// TwinCAT 3 PLC project WeldApp
// ProgramVersion: 3.1.4024.0
// libraries:
//   Tc2_Standard, * (Beckhoff Automation GmbH)
//   Tc2_System, * (Beckhoff Automation GmbH)
//   Tc3_Module, * (Beckhoff Automation GmbH)
//   VisuDialogs, * (System)
// project tree:
//   DUTs/ FixtureInput.TcDUT (not stored), FixtureOutput.TcDUT, Fixture_Clamp.TcDUT
//   / GlobalTextList.TcGTLO, PlcTask.TcTTO, Visualization Manager.TcVMO (not stored)
//   GVLs/ IO.TcGVL, IO_1.TcGVL, IO_1_1.TcGVL, IO_2.TcGVL
//   POUs/ FB_AutoSequence.TcPOU, FB_Clamp.TcPOU, FB_Robot_MH.TcPOU, FB_RollerDoor.TcPOU, FB_ModeManager.TcPOU, FB_Robot.TcPOU, MAIN.TcPOU, FB_Trunnion.TcPOU, FB_TurnTable.TcPOU, TextList_State1.TcTLO, TextList_State2.TcTLO, Visualization.TcVIS
// real-time tasks:
//   TASK PlcTask: cycle T#10ms, priority 20, ADS port 350

CONFIGURATION WeldApp
    RESOURCE PLC ON TwinCAT3
        TASK PlcTask(INTERVAL := T#10ms, PRIORITY := 20);
        PROGRAM MAIN WITH PlcTask : MAIN;
    END_RESOURCE
END_CONFIGURATION

// ---- DUTs/FixtureOutput.TcDUT
TYPE FixtureOutput :
STRUCT
o_CC1_CLAMPING_UNIT1_3_WP:BOOL;
o_CC1_CLAMPING_UNIT1_3_HP:BOOL;
o_CC2_CLAMPING_UNIT2_3_WP:BOOL;
o_CC2_CLAMPING_UNIT2_3_HP:BOOL;
o_CC3_CLAMPING_UNIT3_3_WP:BOOL;
o_CC3_CLAMPING_UNIT3_3_HP:BOOL;
o_CC4_CLAMPING_UNIT4_3_WP:BOOL;
o_CC4_CLAMPING_UNIT4_3_HP:BOOL;
o_CC5_CLAMPING_UNIT5_1_WP:BOOL;
o_CC5_CLAMPING_UNIT5_1_HP:BOOL;
o_CC6_CLAMPING_UNIT6_1_WP:BOOL;
o_CC6_CLAMPING_UNIT6_1_HP:BOOL;
o_RESERVE_1_4:BOOL;
o_RESERVE_1_5:BOOL;
o_RESERVE_1_6:BOOL;
o_RESERVE_1_7:BOOL;
o_RESERVE_2_0:BOOL;
o_RESERVE_2_1:BOOL;
o_RESERVE_2_2:BOOL;
o_RESERVE_2_3:BOOL;
o_RESERVE_2_4:BOOL;
o_RESERVE_2_5:BOOL;
o_RESERVE_2_6:BOOL;
o_RESERVE_2_7:BOOL;
o_RESERVE_3_0:BOOL;
o_RESERVE_3_1:BOOL;
o_RESERVE_3_2:BOOL;
o_RESERVE_3_3:BOOL;
o_RESERVE_3_4:BOOL;
o_RESERVE_3_5:BOOL;
o_RESERVE_3_6:BOOL;
o_RESERVE_3_7:BOOL;

END_STRUCT
END_TYPE

// ---- DUTs/Fixture_Clamp.TcDUT
TYPE Fixture_Clamp :
STRUCT	
	CC1_CloseCmd      : BOOL;
	CC1Done           : BOOL;
    CC2_CloseCmd      : BOOL;
	CC2Done           : BOOL;
	CC3_CloseCmd      : BOOL;
	CC3Done           : BOOL;
    CC4_CloseCmd      : BOOL;
	CC4Done           : BOOL;
	CC5_CloseCmd      : BOOL;
	CC5Done           : BOOL;
    CC6_CloseCmd      : BOOL;
	CC6Done           : BOOL;
	
    CC1_OpenCmd  : BOOL;
    CC2_OpenCmd  : BOOL;
    CC3_OpenCmd  : BOOL;
    CC4_OpenCmd  : BOOL;
    CC5_OpenCmd  : BOOL;
    CC6_OpenCmd  : BOOL;
END_STRUCT
END_TYPE

// ---- GVLs/IO.TcGVL
{attribute 'qualified_only'}
VAR_GLOBAL
	Fixture1Input:FixtureInput;
	Fixture1Output:FixtureOutput;
	Fixture2Input:FixtureInput;
	Fixture2Output:FixtureOutput;
END_VAR

// ---- GVLs/IO_1.TcGVL
{attribute 'qualified_only'}
VAR_GLOBAL
	Fixture1Input:FixtureInput;
	Fixture1Output:FixtureOutput;
	Fixture2Input:FixtureInput;
	Fixture2Output:FixtureOutput;
END_VAR

// ---- GVLs/IO_1_1.TcGVL
{attribute 'qualified_only'}
VAR_GLOBAL
	Fixture1Input:FixtureInput;
	Fixture1Output:FixtureOutput;
	Fixture2Input:FixtureInput;
	Fixture2Output:FixtureOutput;
END_VAR

// ---- GVLs/IO_2.TcGVL
{attribute 'qualified_only'}
VAR_GLOBAL
	Fixture1Input:FixtureInput;
	Fixture1Output:FixtureOutput;
	Fixture2Input:FixtureInput;
	Fixture2Output:FixtureOutput;
END_VAR

// ---- POUs/MAIN.TcPOU
PROGRAM MAIN
VAR
    //=================================================
    // FB INSTANCES
    //=================================================
    ModeMgr    : FB_ModeManager;
    AutoSeq    : FB_AutoSequence;
	
	Fixture_1_CC1     : FB_Clamp;
    Fixture_1_CC2     : FB_Clamp;
	Fixture_1_CC3     : FB_Clamp;
    Fixture_1_CC4     : FB_Clamp;
	Fixture_1_CC5     : FB_Clamp;
	Fixture_1_CC6     : FB_Clamp;
	
	Fixture_2_CC1     : FB_Clamp;
    Fixture_2_CC2     : FB_Clamp;
	Fixture_2_CC3     : FB_Clamp;
    Fixture_2_CC4     : FB_Clamp;
	Fixture_2_CC5     : FB_Clamp;
	Fixture_2_CC6     : FB_Clamp;
	
	RollerDoor1     : FB_RollerDoor;
	RollerDoor2     : FB_RollerDoor;
	
    Trunnion1   : FB_Trunnion;
	Trunnion2   : FB_Trunnion;
	
    Turntable   : FB_Turntable;

    Robot1      : FB_Robot;
	Robot2      : FB_Robot_MH;

    //=================================================
    // HMI INPUTS
    //=================================================
    CycleStart   : BOOL;

    HMI_Auto     : BOOL;
    HMI_Manual   : BOOL;

    PartPresent1 : BOOL;
    PartPresent2 : BOOL;
	
	PartPresent3 : BOOL;
    PartPresent4 : BOOL;
	
    EmergencyStop   : BOOL;   // TRUE = OK
    LightCurtainOK  : BOOL;   // TRUE = OK

    //---------------- Manual Controls ----------------
    Fixture_1_ManCC1Close : BOOL;
    Fixture_1_ManCC1Open  : BOOL;

    Fixture_1_ManCC2Close : BOOL;
    Fixture_1_ManCC2Open  : BOOL;
	
	Fixture_1_ManCC3Close : BOOL;
    Fixture_1_ManCC3Open  : BOOL;

    Fixture_1_ManCC4Close : BOOL;
    Fixture_1_ManCC4Open  : BOOL;
	
	Fixture_1_ManCC5Close : BOOL;
    Fixture_1_ManCC5Open  : BOOL;
	
	Fixture_1_ManCC6Close : BOOL;
    Fixture_1_ManCC6Open  : BOOL;

	Fixture_2_ManCC1Close : BOOL;
    Fixture_2_ManCC1Open  : BOOL;

    Fixture_2_ManCC2Close : BOOL;
    Fixture_2_ManCC2Open  : BOOL;
	
	Fixture_2_ManCC3Close : BOOL;
    Fixture_2_ManCC3Open  : BOOL;

    Fixture_2_ManCC4Close : BOOL;
    Fixture_2_ManCC4Open  : BOOL;
	
	Fixture_2_ManCC5Close : BOOL;
    Fixture_2_ManCC5Open  : BOOL;
	
	Fixture_2_ManCC6Close : BOOL;
    Fixture_2_ManCC6Open  : BOOL;	
	
    ManRollerDoor1Close : BOOL;
    ManRollerDoor1Open  : BOOL;	
	
    ManRollerDoor2Close : BOOL;
    ManRollerDoor2Open  : BOOL;	

    ManTrn10        : BOOL;
    ManTrn150       : BOOL;
	
    ManTrn20        : BOOL;
    ManTrn250       : BOOL;	

    ManTT0         : BOOL;
    ManTT180       : BOOL;

    ManWeld1       : BOOL;
    ManWeld2       : BOOL;

    //=================================================
    // INTERNAL SIGNALS
    //=================================================
    SafetyOK   : BOOL;
    SystemIdle : BOOL;

END_VAR

SafetyOK := EmergencyStop AND LightCurtainOK;

SystemIdle :=
    NOT Trunnion1.Busy AND
	NOT Trunnion2.Busy AND
    NOT Turntable.Busy AND
    NOT Robot1.Busy AND
	NOT Robot2.Busy AND
    NOT Fixture_1_CC1.Busy AND
    NOT Fixture_1_CC2.Busy AND 
	NOT Fixture_1_CC3.Busy AND
    NOT Fixture_1_CC4.Busy AND 
    NOT Fixture_1_CC5.Busy AND
    NOT Fixture_1_CC6.Busy AND
	NOT Fixture_2_CC1.Busy AND
    NOT Fixture_2_CC2.Busy AND 
	NOT Fixture_2_CC3.Busy AND
    NOT Fixture_2_CC4.Busy AND 
    NOT Fixture_2_CC5.Busy AND
    NOT Fixture_2_CC6.Busy;
	
ModeMgr(
    AutoReq    := HMI_Auto,
    ManualReq  := HMI_Manual,
    SafetyOK   := SafetyOK,
    SystemIdle := SystemIdle
);

//Fixture 1
//--------------------------------------------------
// CC1 CONTROL
//--------------------------------------------------
Fixture_1_CC1(
    CloseCmd := ((AutoSeq.Fixture_1_CC1_CloseCmd AND ModeMgr.AutoMode) OR (Fixture_1_ManCC1Close AND ModeMgr.ManualMode)) AND SafetyOK,
    OpenCmd  := ((AutoSeq.Fixture_1_CC1_OpenCmd AND ModeMgr.AutoMode) OR (Fixture_1_ManCC1Open AND ModeMgr.ManualMode)) AND SafetyOK
);
	IO.Fixture1Input.i_CC1_Clamp_1_Sensor_WP:= Fixture_1_CC1.ClosedSim; 
	IO.Fixture1Input.i_CC1_Clamp_2_Sensor_WP:= Fixture_1_CC1.ClosedSim;
	IO.Fixture1Input.i_CC1_Clamp_3_Sensor_WP:= Fixture_1_CC1.ClosedSim;

//--------------------------------------------------
// CC2 CONTROL
//--------------------------------------------------
Fixture_1_CC2(
    CloseCmd := ((AutoSeq.Fixture_1_CC2_CloseCmd AND ModeMgr.AutoMode) OR (Fixture_1_ManCC2Close AND ModeMgr.ManualMode)) AND SafetyOK,
    OpenCmd  := ((AutoSeq.Fixture_1_CC2_OpenCmd AND ModeMgr.AutoMode) OR (Fixture_1_ManCC2Open AND ModeMgr.ManualMode)) AND SafetyOK
);
	IO.Fixture1Input.i_CC2_Clamp_1_Sensor_WP:= Fixture_1_CC2.ClosedSim;
 	IO.Fixture1Input.i_CC2_Clamp_2_Sensor_WP:= Fixture_1_CC2.ClosedSim; 
	IO.Fixture1Input.i_CC2_Clamp_3_Sensor_WP:= Fixture_1_CC2.ClosedSim;

//--------------------------------------------------
// CC3 CONTROL
//--------------------------------------------------
Fixture_1_CC3(
    CloseCmd := ((AutoSeq.Fixture_1_CC3_CloseCmd AND ModeMgr.AutoMode) OR (Fixture_1_ManCC3Close AND ModeMgr.ManualMode)) AND SafetyOK,
    OpenCmd  := ((AutoSeq.Fixture_1_CC3_OpenCmd AND ModeMgr.AutoMode) OR (Fixture_1_ManCC3Open AND ModeMgr.ManualMode)) AND SafetyOK
);
	IO.Fixture1Input.i_CC3_Clamp_1_Sensor_WP:= Fixture_1_CC3.ClosedSim;
	IO.Fixture1Input.i_CC3_Clamp_2_Sensor_WP:= Fixture_1_CC3.ClosedSim;
	IO.Fixture1Input.i_CC3_Clamp_3_Sensor_WP:= Fixture_1_CC3.ClosedSim;

//--------------------------------------------------
// CC4 CONTROL
//--------------------------------------------------
Fixture_1_CC4(
    CloseCmd := ((AutoSeq.Fixture_1_CC4_CloseCmd AND ModeMgr.AutoMode) OR (Fixture_1_ManCC4Close AND ModeMgr.ManualMode)) AND SafetyOK,
    OpenCmd  := ((AutoSeq.Fixture_1_CC4_OpenCmd AND ModeMgr.AutoMode) OR (Fixture_1_ManCC4Open AND ModeMgr.ManualMode)) AND SafetyOK
);
	IO.Fixture1Input.i_CC4_Clamp_1_Sensor_WP:= Fixture_1_CC4.ClosedSim;
	IO.Fixture1Input.i_CC4_Clamp_2_Sensor_WP:= Fixture_1_CC4.ClosedSim;
	IO.Fixture1Input.i_CC4_Clamp_3_Sensor_WP:= Fixture_1_CC4.ClosedSim;

//--------------------------------------------------
// CC5 CONTROL
//--------------------------------------------------
Fixture_1_CC5(
    CloseCmd := ((AutoSeq.Fixture_1_CC5_CloseCmd AND ModeMgr.AutoMode) OR (Fixture_1_ManCC5Close AND ModeMgr.ManualMode)) AND SafetyOK,
    OpenCmd  := ((AutoSeq.Fixture_1_CC5_OpenCmd AND ModeMgr.AutoMode) OR (Fixture_1_ManCC5Open AND ModeMgr.ManualMode)) AND SafetyOK
);
    IO.Fixture1Input.i_CC5_Clamp_1_Sensor_WP:= Fixture_1_CC5.ClosedSim;

//--------------------------------------------------
// CC6 CONTROL
//--------------------------------------------------
Fixture_1_CC6(
    CloseCmd := ((AutoSeq.Fixture_1_CC6_CloseCmd AND ModeMgr.AutoMode) OR (Fixture_1_ManCC6Close AND ModeMgr.ManualMode)) AND SafetyOK,
    OpenCmd  := ((AutoSeq.Fixture_1_CC6_OpenCmd AND ModeMgr.AutoMode) OR (Fixture_1_ManCC6Open AND ModeMgr.ManualMode)) AND SafetyOK
);
	IO.Fixture1Input.i_CC6_Clamp_1_Sensor_WP:= Fixture_1_CC6.ClosedSim;
	
//Fixture 2
//--------------------------------------------------
// CC1 CONTROL
//--------------------------------------------------
Fixture_2_CC1(
    CloseCmd := ((AutoSeq.Fixture_2_CC1_CloseCmd AND ModeMgr.AutoMode) OR (Fixture_2_ManCC1Close AND ModeMgr.ManualMode)) AND SafetyOK,
    OpenCmd  := ((AutoSeq.Fixture_2_CC1_OpenCmd AND ModeMgr.AutoMode) OR (Fixture_2_ManCC1Open AND ModeMgr.ManualMode)) AND SafetyOK
);
	IO.Fixture2Input.i_CC1_Clamp_1_Sensor_WP:= Fixture_2_CC1.ClosedSim;
	IO.Fixture2Input.i_CC1_Clamp_2_Sensor_WP:= Fixture_2_CC1.ClosedSim;
	IO.Fixture2Input.i_CC1_Clamp_3_Sensor_WP:= Fixture_2_CC1.ClosedSim;
	
//--------------------------------------------------
// CC2 CONTROL
//--------------------------------------------------
Fixture_2_CC2(
    CloseCmd := ((AutoSeq.Fixture_2_CC2_CloseCmd AND ModeMgr.AutoMode) OR (Fixture_2_ManCC2Close AND ModeMgr.ManualMode)) AND SafetyOK,
    OpenCmd  := ((AutoSeq.Fixture_2_CC2_OpenCmd AND ModeMgr.AutoMode) OR (Fixture_2_ManCC2Open AND ModeMgr.ManualMode)) AND SafetyOK
);
	IO.Fixture2Input.i_CC2_Clamp_1_Sensor_WP:= Fixture_2_CC2.ClosedSim;
	IO.Fixture2Input.i_CC2_Clamp_2_Sensor_WP:= Fixture_2_CC2.ClosedSim;
	IO.Fixture2Input.i_CC2_Clamp_3_Sensor_WP:= Fixture_2_CC2.ClosedSim;

//--------------------------------------------------
// CC3 CONTROL
//--------------------------------------------------
Fixture_2_CC3(
    CloseCmd := ((AutoSeq.Fixture_2_CC3_CloseCmd AND ModeMgr.AutoMode) OR (Fixture_2_ManCC3Close AND ModeMgr.ManualMode)) AND SafetyOK,
    OpenCmd  := ((AutoSeq.Fixture_2_CC3_OpenCmd AND ModeMgr.AutoMode) OR (Fixture_2_ManCC3Open AND ModeMgr.ManualMode)) AND SafetyOK
);
	IO.Fixture2Input.i_CC3_Clamp_1_Sensor_WP:= Fixture_2_CC3.ClosedSim;
	IO.Fixture2Input.i_CC3_Clamp_2_Sensor_WP:= Fixture_2_CC3.ClosedSim;
	IO.Fixture2Input.i_CC3_Clamp_3_Sensor_WP:= Fixture_2_CC3.ClosedSim;
 
//--------------------------------------------------
// CC4 CONTROL
//--------------------------------------------------
Fixture_2_CC4(
    CloseCmd := ((AutoSeq.Fixture_2_CC4_CloseCmd AND ModeMgr.AutoMode) OR (Fixture_2_ManCC4Close AND ModeMgr.ManualMode)) AND SafetyOK,
    OpenCmd  := ((AutoSeq.Fixture_2_CC4_OpenCmd AND ModeMgr.AutoMode) OR (Fixture_2_ManCC4Open AND ModeMgr.ManualMode)) AND SafetyOK
);
	IO.Fixture2Input.i_CC4_Clamp_1_Sensor_WP := Fixture_2_CC4.ClosedSim;
	IO.Fixture2Input.i_CC4_Clamp_2_Sensor_WP := Fixture_2_CC4.ClosedSim;
	IO.Fixture2Input.i_CC4_Clamp_3_Sensor_WP := Fixture_2_CC4.ClosedSim;

//--------------------------------------------------
// CC5 CONTROL
//--------------------------------------------------
Fixture_2_CC5(
    CloseCmd := ((AutoSeq.Fixture_2_CC5_CloseCmd AND ModeMgr.AutoMode) OR (Fixture_2_ManCC5Close AND ModeMgr.ManualMode)) AND SafetyOK,
    OpenCmd  := ((AutoSeq.Fixture_2_CC5_OpenCmd AND ModeMgr.AutoMode) OR (Fixture_2_ManCC5Open AND ModeMgr.ManualMode)) AND SafetyOK
);
	IO.Fixture2Input.i_CC5_Clamp_1_Sensor_WP:= Fixture_2_CC5.ClosedSim;

//--------------------------------------------------
// CC6 CONTROL
//--------------------------------------------------
Fixture_2_CC6(
    CloseCmd := ((AutoSeq.Fixture_2_CC6_CloseCmd AND ModeMgr.AutoMode) OR (Fixture_2_ManCC6Close AND ModeMgr.ManualMode)) AND SafetyOK,
    OpenCmd  := ((AutoSeq.Fixture_2_CC6_OpenCmd AND ModeMgr.AutoMode) OR (Fixture_2_ManCC6Open AND ModeMgr.ManualMode)) AND SafetyOK
);
	IO.Fixture2Input.i_CC6_Clamp_1_Sensor_WP:= Fixture_2_CC6.ClosedSim;	

//--------------------------------------------------
// ROLLER DOOR CONTROL
//--------------------------------------------------
RollerDoor1(
    CloseCmd := ((AutoSeq.RollerDoor1CloseCmd AND ModeMgr.AutoMode) OR (ManRollerDoor1Close AND ModeMgr.ManualMode)) AND SafetyOK,
    OpenCmd  := ((AutoSeq.RollerDoor1OpenCmd AND ModeMgr.AutoMode) OR (ManRollerDoor1Open AND ModeMgr.ManualMode)) AND SafetyOK
);

RollerDoor2(
    CloseCmd := ((AutoSeq.RollerDoor2CloseCmd AND ModeMgr.AutoMode) OR (ManRollerDoor2Close AND ModeMgr.ManualMode)) AND SafetyOK,
    OpenCmd  := ((AutoSeq.RollerDoor2OpenCmd AND ModeMgr.AutoMode) OR (ManRollerDoor2Open AND ModeMgr.ManualMode)) AND SafetyOK
);

//--------------------------------------------------
// TRUNNION CONTROL
//--------------------------------------------------
Trunnion1(
    To0  := ((AutoSeq.Trunnion1To0 AND ModeMgr.AutoMode) OR (ManTrn10 AND ModeMgr.ManualMode)) AND SafetyOK,
    To50 := ((AutoSeq.Trunnion1To50 AND ModeMgr.AutoMode) OR (ManTrn150 AND ModeMgr.ManualMode)) AND SafetyOK
);

Trunnion2(
    To0  := ((AutoSeq.Trunnion2To0 AND ModeMgr.AutoMode) OR (ManTrn20 AND ModeMgr.ManualMode)) AND SafetyOK,
    To50 := ((AutoSeq.Trunnion2To50 AND ModeMgr.AutoMode) OR (ManTrn250 AND ModeMgr.ManualMode)) AND SafetyOK
);


//--------------------------------------------------
// TURNTABLE CONTROL
//--------------------------------------------------
Turntable(
    To180 := ((AutoSeq.Turn180 AND ModeMgr.AutoMode) OR (ManTT180 AND ModeMgr.ManualMode)) AND SafetyOK,
    To0   := ((AutoSeq.TurnTo0 AND ModeMgr.AutoMode) OR (ManTT0 AND ModeMgr.ManualMode)) AND SafetyOK
);


//--------------------------------------------------
// WELD ROBOT CONTROL
//--------------------------------------------------
Robot1(
    StartWeld1 := ((AutoSeq.RobotWeldStart1 AND ModeMgr.AutoMode) OR (ManWeld1 AND ModeMgr.ManualMode)) AND SafetyOK,
    StartWeld2 := ((AutoSeq.RobotWeldStart2 AND ModeMgr.AutoMode) OR (ManWeld2 AND ModeMgr.ManualMode)) AND SafetyOK
);

//--------------------------------------------------
// MH ROBOT CONTROL
//--------------------------------------------------
Robot2(
    ClearToPick1 := ((AutoSeq.RobotClearPick1 AND ModeMgr.AutoMode) OR (ManWeld1 AND ModeMgr.ManualMode)) AND SafetyOK,
    ClearToPick2 := ((AutoSeq.RobotClearPick2 AND ModeMgr.AutoMode) OR (ManWeld2 AND ModeMgr.ManualMode)) AND SafetyOK
);

//--------------------------------------------------
// AUTO SEQUENCE CONTROL (MAIN LOGIC)
//--------------------------------------------------
AutoSeq(
    CycleStart    := CycleStart AND ModeMgr.AutoMode AND SafetyOK,

    AutoMode      := ModeMgr.AutoMode,

    PartPresent1  := IO.Fixture1Input.i_PART_CONTROL_B1 AND 
					 IO.Fixture1Input.i_PART_CONTROL_B2 AND 
					 IO.Fixture1Input.i_PART_CONTROL_B3 AND 
 					 IO.Fixture1Input.i_PART_CONTROL_B4 AND  
				     IO.Fixture1Input.i_PART_CONTROL_B5 AND 
             		 IO.Fixture1Input.i_PART_CONTROL_B6 AND 
					 IO.Fixture1Input.i_PART_CONTROL_B7,
					 
    PartPresent2  := IO.Fixture1Input.i_PART_CONTROL_B8 AND 
					 IO.Fixture1Input.i_PART_CONTROL_B9 AND 
					 IO.Fixture1Input.i_PART_CONTROL_B10 AND 
 					 IO.Fixture1Input.i_PART_CONTROL_B11 AND  
				     IO.Fixture1Input.i_PART_CONTROL_B12 AND 
             		 IO.Fixture1Input.i_PART_CONTROL_B13 AND 
					 IO.Fixture1Input.i_PART_CONTROL_B14,
	
	PartPresent3  := IO.Fixture2Input.i_PART_CONTROL_B1 AND 
					 IO.Fixture2Input.i_PART_CONTROL_B2 AND 
					 IO.Fixture2Input.i_PART_CONTROL_B3 AND 
 					 IO.Fixture2Input.i_PART_CONTROL_B4 AND  
				     IO.Fixture2Input.i_PART_CONTROL_B5 AND 
             		 IO.Fixture2Input.i_PART_CONTROL_B6 AND 
					 IO.Fixture2Input.i_PART_CONTROL_B7,
					 
    PartPresent4  := IO.Fixture2Input.i_PART_CONTROL_B8 AND 
					 IO.Fixture2Input.i_PART_CONTROL_B9 AND 
					 IO.Fixture2Input.i_PART_CONTROL_B10 AND 
 					 IO.Fixture2Input.i_PART_CONTROL_B11 AND  
				     IO.Fixture2Input.i_PART_CONTROL_B12 AND 
             		 IO.Fixture2Input.i_PART_CONTROL_B13 AND 
					 IO.Fixture2Input.i_PART_CONTROL_B14,

    Fixture_1_CC1Done    := Fixture_1_CC1.Done,
    Fixture_1_CC2Done    := Fixture_1_CC2.Done,
    Fixture_1_CC3Done    := Fixture_1_CC3.Done,	
	Fixture_1_CC4Done    := Fixture_1_CC4.Done,
	Fixture_1_CC5Done    := Fixture_1_CC5.Done,
	Fixture_1_CC6Done    := Fixture_1_CC6.Done,
	
    Fixture_2_CC1Done    := Fixture_2_CC1.Done,
    Fixture_2_CC2Done    := Fixture_2_CC2.Done,
    Fixture_2_CC3Done    := Fixture_2_CC3.Done,	
	Fixture_2_CC4Done    := Fixture_2_CC4.Done,
	Fixture_2_CC5Done    := Fixture_2_CC5.Done,
	Fixture_2_CC6Done    := Fixture_2_CC6.Done,	
	
	RollerDoor1Done    := RollerDoor1.Done,
    RollerDoor2Done    := RollerDoor2.Done,

    TurntableAt0   := Turntable.At0,
    TurntableAt180 := Turntable.At180,

    WeldComplete1 := Robot1.WeldDone1,
    WeldComplete2 := Robot1.WeldDone2,
	
	PickComplete1 := Robot2.Pick1Done1,
    PickComplete2 := Robot2.Pick2Done2,

    Trunnion1At0   := Trunnion1.At0,
    Trunnion1At50  := Trunnion1.At50,
	
    Trunnion2At0   := Trunnion2.At0,
    Trunnion2At50  := Trunnion2.At50	
);

    IO.Fixture1Input.i_PART_CONTROL_B1:=PartPresent1;
	IO.Fixture1Input.i_PART_CONTROL_B2:=PartPresent1;
	IO.Fixture1Input.i_PART_CONTROL_B3:=PartPresent1;
 	IO.Fixture1Input.i_PART_CONTROL_B4:=PartPresent1;
	IO.Fixture1Input.i_PART_CONTROL_B5:=PartPresent1;
    IO.Fixture1Input.i_PART_CONTROL_B6:=PartPresent1;
	IO.Fixture1Input.i_PART_CONTROL_B7:=PartPresent1;
					 
    IO.Fixture1Input.i_PART_CONTROL_B8:=PartPresent2;
	IO.Fixture1Input.i_PART_CONTROL_B9:=PartPresent2;
	IO.Fixture1Input.i_PART_CONTROL_B10:=PartPresent2;
 	IO.Fixture1Input.i_PART_CONTROL_B11:=PartPresent2;
	IO.Fixture1Input.i_PART_CONTROL_B12:=PartPresent2;
    IO.Fixture1Input.i_PART_CONTROL_B13:=PartPresent2;
	IO.Fixture1Input.i_PART_CONTROL_B14:=PartPresent2;
	
    IO.Fixture2Input.i_PART_CONTROL_B1:=PartPresent3;
	IO.Fixture2Input.i_PART_CONTROL_B2:=PartPresent3;
	IO.Fixture2Input.i_PART_CONTROL_B3:=PartPresent3;
 	IO.Fixture2Input.i_PART_CONTROL_B4:=PartPresent3;
	IO.Fixture2Input.i_PART_CONTROL_B5:=PartPresent3;
    IO.Fixture2Input.i_PART_CONTROL_B6:=PartPresent3;
	IO.Fixture2Input.i_PART_CONTROL_B7:=PartPresent3;
					 
    IO.Fixture2Input.i_PART_CONTROL_B8:=PartPresent4;
	IO.Fixture2Input.i_PART_CONTROL_B9:=PartPresent4;
	IO.Fixture2Input.i_PART_CONTROL_B10:=PartPresent4;
 	IO.Fixture2Input.i_PART_CONTROL_B11:=PartPresent4;
	IO.Fixture2Input.i_PART_CONTROL_B12:=PartPresent4;
    IO.Fixture2Input.i_PART_CONTROL_B13:=PartPresent4;
	IO.Fixture2Input.i_PART_CONTROL_B14:=PartPresent4;

END_PROGRAM

// ---- POUs/FB_ModeManager.TcPOU
FUNCTION_BLOCK FB_ModeManager
VAR_INPUT
    AutoReq      : BOOL;   // Request Auto mode (HMI)
    ManualReq    : BOOL;   // Request Manual mode (HMI)

    SafetyOK     : BOOL;   // From safety logic
    SystemIdle   : BOOL;   // TRUE when machine is safe (no motion)
END_VAR

VAR_OUTPUT
    AutoMode     : BOOL;
    ManualMode   : BOOL;

    ModeActive   : BOOL;   // Any mode active
END_VAR

VAR
    State : INT := 0;

END_VAR

CASE State OF

//--------------------------------------------------
// 0: NO MODE SELECTED
//--------------------------------------------------
0:
    AutoMode := FALSE;
    ManualMode := FALSE;
    ModeActive := FALSE;

    // Select Manual first (safe default)
    IF ManualReq AND SafetyOK THEN
        State := 20;

    ELSIF AutoReq AND SafetyOK THEN
        State := 10;
    END_IF


//--------------------------------------------------
// 10: AUTO MODE ACTIVE
//--------------------------------------------------
10:
    AutoMode := TRUE;
    ManualMode := FALSE;
    ModeActive := TRUE;

    // Switch to Manual only when safe
    IF ManualReq AND SystemIdle AND SafetyOK THEN
        State := 20;
    END_IF

    // Drop mode if safety lost
    IF NOT SafetyOK THEN
        State := 0;
    END_IF


//--------------------------------------------------
// 20: MANUAL MODE ACTIVE
//--------------------------------------------------
20:
    AutoMode := FALSE;
    ManualMode := TRUE;
    ModeActive := TRUE;

    // Switch to Auto only when safe
    IF AutoReq AND SystemIdle AND SafetyOK THEN
	   State := 10;
    END_IF

    // Drop mode if safety lost
    IF NOT SafetyOK THEN
        State := 0;
    END_IF

END_CASE

END_FUNCTION_BLOCK

// ---- POUs/FB_AutoSequence.TcPOU
FUNCTION_BLOCK FB_AutoSequence
VAR_INPUT
    CycleStart     : BOOL;
    AutoMode       : BOOL;

    PartPresent1   : BOOL;
    PartPresent2   : BOOL;
	
	PartPresent3   : BOOL;
    PartPresent4   : BOOL;
	

	Fixture_1_CC1Done           : BOOL;
	Fixture_1_CC2Done           : BOOL;
	Fixture_1_CC3Done           : BOOL;
	Fixture_1_CC4Done           : BOOL;
	Fixture_1_CC5Done           : BOOL;
	Fixture_1_CC6Done           : BOOL;
	
	Fixture_1_CC1_CloseCmd      : BOOL;
    Fixture_1_CC2_CloseCmd      : BOOL;
	Fixture_1_CC3_CloseCmd      : BOOL;
    Fixture_1_CC4_CloseCmd      : BOOL;
	Fixture_1_CC5_CloseCmd      : BOOL;
    Fixture_1_CC6_CloseCmd      : BOOL;
	
    Fixture_1_CC1_OpenCmd  : BOOL;
    Fixture_1_CC2_OpenCmd  : BOOL;
    Fixture_1_CC3_OpenCmd  : BOOL;
    Fixture_1_CC4_OpenCmd  : BOOL;
    Fixture_1_CC5_OpenCmd  : BOOL;
    Fixture_1_CC6_OpenCmd  : BOOL;
	
	Fixture_2_CC1Done           : BOOL;
	Fixture_2_CC2Done           : BOOL;
	Fixture_2_CC3Done           : BOOL;
	Fixture_2_CC4Done           : BOOL;
	Fixture_2_CC5Done           : BOOL;
	Fixture_2_CC6Done           : BOOL;
	
	Fixture_2_CC1_CloseCmd      : BOOL;
    Fixture_2_CC2_CloseCmd      : BOOL;
	Fixture_2_CC3_CloseCmd      : BOOL;
    Fixture_2_CC4_CloseCmd      : BOOL;
	Fixture_2_CC5_CloseCmd      : BOOL;
    Fixture_2_CC6_CloseCmd      : BOOL;
	
    Fixture_2_CC1_OpenCmd  : BOOL;
    Fixture_2_CC2_OpenCmd  : BOOL;
    Fixture_2_CC3_OpenCmd  : BOOL;
    Fixture_2_CC4_OpenCmd  : BOOL;
    Fixture_2_CC5_OpenCmd  : BOOL;
    Fixture_2_CC6_OpenCmd  : BOOL;

	RollerDoor1Done	   :BOOL;
	RollerDoor2Done	   :BOOL;

    TurntableAt0   : BOOL;
    TurntableAt180 : BOOL;

    WeldComplete1  : BOOL;
    WeldComplete2  : BOOL;
	
    PickComplete1  : BOOL;
    PickComplete2  : BOOL;

    Trunnion1At0    : BOOL;
    Trunnion1At50   : BOOL;
	
	Trunnion2At0    : BOOL;
    Trunnion2At50   : BOOL;
END_VAR

VAR_OUTPUT
    // Clamp commands
	
	// Door commands
	RollerDoor1CloseCmd : BOOL;
	RollerDoor1OpenCmd  : BOOL;
	
	RollerDoor2CloseCmd : BOOL;
	RollerDoor2OpenCmd  : BOOL;
	
    // Motion commands
    Trunnion1To0    : BOOL;
    Trunnion1To50   : BOOL;

    Trunnion2To0    : BOOL;
    Trunnion2To50   : BOOL;
	
    Turn180        : BOOL;
    TurnTo0        : BOOL;

    // Robot commands
    RobotWeldStart1    : BOOL;
    RobotWeldStart2    : BOOL;
	RobotClearPick1    : BOOL;
    RobotClearPick2    : BOOL;
END_VAR

VAR
    State1 : INT := 0;
	State2 : INT := 0;
END_VAR

//--------------------------------------------------
// RESET OUTPUTS EVERY CYCLE
//--------------------------------------------------
Fixture_1_CC1_CloseCmd := FALSE;
Fixture_1_CC2_CloseCmd := FALSE;
Fixture_1_CC3_CloseCmd := FALSE;
Fixture_1_CC4_CloseCmd := FALSE;
Fixture_1_CC5_CloseCmd := FALSE;
Fixture_1_CC6_CloseCmd := FALSE;

Fixture_1_CC1_OpenCmd := FALSE;
Fixture_1_CC2_OpenCmd := FALSE;
Fixture_1_CC3_OpenCmd := FALSE;
Fixture_1_CC4_OpenCmd := FALSE;
Fixture_1_CC5_OpenCmd := FALSE;
Fixture_1_CC6_OpenCmd := FALSE;

Fixture_2_CC1_CloseCmd := FALSE;
Fixture_2_CC2_CloseCmd := FALSE;
Fixture_2_CC3_CloseCmd := FALSE;
Fixture_2_CC4_CloseCmd := FALSE;
Fixture_2_CC5_CloseCmd := FALSE;
Fixture_2_CC6_CloseCmd := FALSE;

Fixture_2_CC1_OpenCmd := FALSE;
Fixture_2_CC2_OpenCmd := FALSE;
Fixture_2_CC3_OpenCmd := FALSE;
Fixture_2_CC4_OpenCmd := FALSE;
Fixture_2_CC5_OpenCmd := FALSE;
Fixture_2_CC6_OpenCmd := FALSE;

RollerDoor1CloseCmd := FALSE;
RollerDoor1OpenCmd  := FALSE;

RollerDoor2CloseCmd := FALSE;
RollerDoor2OpenCmd  := FALSE;

Trunnion1To0 := FALSE;
Trunnion1To50 := FALSE;
Trunnion2To0 := FALSE;
Trunnion2To50 := FALSE;

Turn180 := FALSE;
TurnTo0 := FALSE;

RobotWeldStart1 := FALSE;
RobotWeldStart2 := FALSE;
RobotClearPick1 := FALSE;
RobotClearPick2 := FALSE;

//--------------------------------------------------
// SEQUENCE LOGIC
//--------------------------------------------------
CASE State1 OF

//--------------------------------------------------
// 0: OPEN DOOR
//--------------------------------------------------
0:
    IF TurntableAt0 AND NOT PartPresent1 THEN
	RollerDoor1OpenCmd := TRUE;
	END_IF

    IF RollerDoor1Done AND TurntableAt0 AND NOT PartPresent1 THEN
        State1 := 10;
    END_IF
	
//--------------------------------------------------
// 10: WAIT FOR START + PART 1
//--------------------------------------------------
10:
    IF AutoMode AND CycleStart AND PartPresent1  THEN
        State1 := 20;
    END_IF
	
//--------------------------------------------------
// 20: CLOSE DOOR
//--------------------------------------------------
20:
    RollerDoor1CloseCmd := TRUE;

    IF RollerDoor1Done THEN
        State1 := 30;
    END_IF

//--------------------------------------------------
// 30: CLOSE CLAMP CC1 CC3 CC5
//--------------------------------------------------
30:
    Fixture_1_CC1_CloseCmd := TRUE;
	Fixture_1_CC3_CloseCmd := TRUE;
	Fixture_1_CC5_CloseCmd := TRUE;
	

    IF Fixture_1_CC1Done AND Fixture_1_CC3Done AND Fixture_1_CC5Done THEN
        State1 := 40;
    END_IF

//--------------------------------------------------
// 40: MOVE TRUNNION TO 50 DEG
//--------------------------------------------------
40:
    Trunnion1To50 := TRUE;

    IF Trunnion1At50 THEN
        State1 := 50;
    END_IF
	
//--------------------------------------------------
// 50: OPEN DOOR
//--------------------------------------------------
50:
    RollerDoor1OpenCmd := TRUE;

    IF RollerDoor1Done THEN
        State1 := 60;
    END_IF


//--------------------------------------------------
// 60: WAIT FOR PART 2
//--------------------------------------------------
60:
    IF PartPresent2 AND CycleStart AND Trunnion1At50 THEN
        State1 := 70;
    END_IF

//--------------------------------------------------
// 70: CLOSE CLAMP CC2 CC4 CC6
//--------------------------------------------------
70:
    Fixture_1_CC2_CloseCmd := TRUE;
	Fixture_1_CC4_CloseCmd := TRUE;
	Fixture_1_CC6_CloseCmd := TRUE;

    IF Fixture_1_CC2Done AND Fixture_1_CC4Done AND Fixture_1_CC6Done THEN
        State1 := 80;
    END_IF
	
//--------------------------------------------------
// 80: CLOSE DOOR
//--------------------------------------------------
80:
    RollerDoor1CloseCmd := TRUE;

    IF RollerDoor1Done THEN
        State1 := 90;
    END_IF


//--------------------------------------------------
// 90: TRUNNION 1 BACK TO 0 DEG
//--------------------------------------------------
90:
    Trunnion1To0 := TRUE;

    IF Trunnion1At0 THEN
        State1 := 100;
    END_IF


//--------------------------------------------------
// 100: TURN TABLE TO 180 DEG (WELD STATION)
//--------------------------------------------------
100:
	IF TurntableAt0 AND PartPresent1 AND PartPresent2 AND Trunnion1At0 THEN
    Turn180 := TRUE;
	END_IF
	
 	IF TurntableAt180 THEN
 	State1 := 110;
	END_IF
	ELSE TurntableAt180:=FALSE;
      
//--------------------------------------------------
// 110: ROBOT WELD 1
//--------------------------------------------------
110:
    RobotWeldStart1 := TRUE;

    IF WeldComplete1 THEN
        State1 := 120;
    END_IF
	
//--------------------------------------------------
// 120: RETURN TRUNNION1 TO 50
//--------------------------------------------------
120:
    Trunnion1To50 := TRUE;

    IF Trunnion1At50 THEN
        State1 := 130;
    END_IF

//--------------------------------------------------
// 130: ROBOT WELD 2
//--------------------------------------------------
130:
    RobotWeldStart2 := TRUE;

    IF WeldComplete2 THEN
        State1 := 140;
    END_IF


//--------------------------------------------------
// 140: OPEN CLAMP CC1 CC3 CC5 
//--------------------------------------------------
140:
	IF PartPresent2 AND TurntableAt180 AND Trunnion1At50 THEN
    Fixture_1_CC1_OpenCmd := TRUE;
	Fixture_1_CC3_OpenCmd := TRUE;
	Fixture_1_CC5_OpenCmd := TRUE;
	END_IF

    IF Fixture_1_CC1Done AND Fixture_1_CC3Done AND Fixture_1_CC5Done  THEN
        State1 := 150;
    END_IF
	
//--------------------------------------------------
// 150: ROBOT PICK 1
//--------------------------------------------------
150:
    RobotClearPick1 := TRUE;

    IF PickComplete1 THEN
        State1 := 160;
    END_IF	
	
//--------------------------------------------------
// 160: RETURN TRUNNION TO 0
//--------------------------------------------------
160:
    Trunnion1To0 := TRUE;

    IF Trunnion1At0 THEN
        State1 := 170;
    END_IF
	
//--------------------------------------------------
// 170: OPEN CLAMP CC2 CC4 CC6 
//--------------------------------------------------
170:
	IF PartPresent1 AND TurntableAt180 AND Trunnion1At0 THEN
    Fixture_1_CC2_OpenCmd := TRUE;
	Fixture_1_CC4_OpenCmd := TRUE;
	Fixture_1_CC6_OpenCmd := TRUE;
	END_IF

    IF Fixture_1_CC2Done AND Fixture_1_CC4Done AND Fixture_1_CC6Done THEN
        State1 := 180;
    END_IF
	
//--------------------------------------------------
// 180: ROBOT PICK 2
//--------------------------------------------------
180:
    RobotClearPick2 := TRUE;

    IF PickComplete2 THEN
        State1 := 0;
    END_IF

END_CASE



//--------------------------------------------------
// SEQUENCE LOGIC
//--------------------------------------------------
CASE State2 OF

//--------------------------------------------------
// 0: OPEN DOOR
//--------------------------------------------------
0:
    IF TurntableAt180 AND NOT PartPresent3 THEN
	RollerDoor1OpenCmd := TRUE;
	END_IF

    IF RollerDoor1Done AND TurntableAt180 AND NOT PartPresent3 THEN
        State2 := 10;
    END_IF


//--------------------------------------------------
// 10: WAIT FOR START + PART 3
//--------------------------------------------------
10:
	IF AutoMode AND CycleStart AND PartPresent3  THEN
        State2 := 20;
    END_IF

//--------------------------------------------------
// 20: DOOR CLOSE
//--------------------------------------------------
20:
	RollerDoor1CloseCmd := TRUE;

    IF RollerDoor1Done THEN
        State2 := 30;
    END_IF
	
//--------------------------------------------------
// 30: CLOSE CLAMP CC1 CC3 CC5
//--------------------------------------------------
30:
    Fixture_2_CC1_CloseCmd := TRUE;
	Fixture_2_CC3_CloseCmd := TRUE;
	Fixture_2_CC5_CloseCmd := TRUE;

    IF Fixture_2_CC1Done AND Fixture_2_CC3Done AND Fixture_2_CC5Done THEN
        State2 := 40;
    END_IF
	
	
//--------------------------------------------------
// 40: MOVE TRUNNION2 TO 50 DEG
//--------------------------------------------------
40:
    Trunnion2To50 := TRUE;

    IF Trunnion2At50 THEN
        State2 := 50;
    END_IF
	
//--------------------------------------------------
// 50: OPEN DOOR
//--------------------------------------------------
50:
	RollerDoor1OpenCmd := TRUE;

    IF RollerDoor1Done THEN
        State2 := 60;
    END_IF	

//--------------------------------------------------
// 60: WAIT FOR PART 4
//--------------------------------------------------
60:
    IF PartPresent4 AND CycleStart THEN
        State2 := 70;
    END_IF
	
//--------------------------------------------------
// 70: DOOR CLOSE
//--------------------------------------------------
70:
	RollerDoor1CloseCmd := TRUE;

    IF RollerDoor1Done THEN
       State2 := 80;
    END_IF

//--------------------------------------------------
// 80: CLOSE CLAMP 4
//--------------------------------------------------
80:
    Fixture_2_CC2_CloseCmd := TRUE;
	Fixture_2_CC4_CloseCmd := TRUE;
	Fixture_2_CC6_CloseCmd := TRUE;

    IF Fixture_2_CC2Done AND Fixture_2_CC4Done AND Fixture_2_CC6Done THEN
        State2 := 90;
    END_IF
	

//--------------------------------------------------
// 90: TRUNNION2 BACK TO 0 DEG
//--------------------------------------------------
90:
    Trunnion2To0 := TRUE;

    IF Trunnion2At0 THEN
        State2 := 100;
    END_IF


//--------------------------------------------------
// 100: TURN TABLE TO 0 DEG (WELD STATION)
//--------------------------------------------------
100:
	IF TurntableAt180 AND NOT( PartPresent1 AND PartPresent2) AND PartPresent3 AND PartPresent4 THEN
    TurnTo0 := TRUE;
	END_IF
	
 	IF TurntableAt0 THEN
 	State2 := 110;
	END_IF
	
      
//--------------------------------------------------
// 110: ROBOT WELD 1
//--------------------------------------------------
110:
    RobotWeldStart1 := TRUE;

    IF WeldComplete1 THEN
        State2 := 120;
    END_IF
	
//--------------------------------------------------
// 120: TRUNNION2 GO TO 50 DEG
//--------------------------------------------------
120:
    Trunnion2To50 := TRUE;

    IF Trunnion2At50 THEN
        State2 := 130;
    END_IF
	
//--------------------------------------------------
// 130: ROBOT WELD 2
//--------------------------------------------------
130:
    RobotWeldStart2 := TRUE;

    IF WeldComplete2 THEN
        State2 := 140;
    END_IF
	
//--------------------------------------------------
// 140: OPEN CLAMP 4
//--------------------------------------------------
140:
	IF PartPresent4 AND TurntableAt0 AND Trunnion1At0 THEN
    Fixture_2_CC2_OpenCmd := TRUE;
	Fixture_2_CC4_OpenCmd := TRUE;
	Fixture_2_CC6_OpenCmd := TRUE;
	END_IF

	IF Fixture_2_CC2Done AND Fixture_2_CC4Done AND Fixture_2_CC6Done  THEN
		PartPresent4:=FALSE;
        State2 := 150;
    END_IF
	
//--------------------------------------------------
// 150: ROBOT PICK 1
//--------------------------------------------------
150:
    RobotClearPick1 := TRUE;

    IF PickComplete1 THEN
        State2 := 160;
    END_IF		

//--------------------------------------------------
// 160: TRUNNION2 BACK TO 0 DEG
//--------------------------------------------------
160:
    Trunnion2To0 := TRUE;

    IF Trunnion2At0 THEN
        State2 := 170;
    END_IF
	
//--------------------------------------------------
// 170: OPEN CLAMP 3
//--------------------------------------------------
170:
	
	IF PartPresent3 AND TurntableAt0 AND Trunnion1At0 THEN
    Fixture_2_CC1_OpenCmd := TRUE;
	Fixture_2_CC3_OpenCmd := TRUE;
	Fixture_2_CC5_OpenCmd := TRUE;
	END_IF

    IF Fixture_2_CC1Done AND Fixture_2_CC3Done AND Fixture_2_CC5Done THEN
		PartPresent3:=FALSE;
        State2 := 180;
    END_IF
	
//--------------------------------------------------
// 180: ROBOT PICK 2
//--------------------------------------------------
180:
    RobotClearPick2 := TRUE;

    IF PickComplete2 THEN
        State2 := 0;
    END_IF
END_CASE

END_FUNCTION_BLOCK

// ---- POUs/FB_Clamp.TcPOU
FUNCTION_BLOCK FB_Clamp
VAR_INPUT
    CloseCmd   : BOOL;
    OpenCmd    : BOOL;
END_VAR

VAR_OUTPUT
    CloseOut   : BOOL;
    OpenOut    : BOOL;
    Done       : BOOL;
    Busy       : BOOL;
    ClosedSim  : BOOL;
    OpenedSim  : BOOL;
END_VAR

VAR
    State   : INT := 0;
    tClose  : TON;
    tOpen   : TON;
END_VAR

CASE State OF

0: // Idle
    Done := FALSE;
    Busy := FALSE;
    CloseOut := FALSE;
    OpenOut := FALSE;

    tClose(IN := FALSE);
    tOpen(IN := FALSE);

    IF CloseCmd THEN
        State := 10;
    ELSIF OpenCmd THEN
        State := 20;
    END_IF


10: // Closing
    Busy := TRUE;
    CloseOut := TRUE;

    tClose(IN := TRUE, PT := T#3s);

    IF tClose.Q THEN
        CloseOut := FALSE;
        Busy := FALSE;
        Done := TRUE;
        ClosedSim := TRUE;
        OpenedSim := FALSE;
        tClose(IN := FALSE);
        State := 0;
    END_IF


20: // Opening
    Busy := TRUE;
    OpenOut := TRUE;

    tOpen(IN := TRUE, PT := T#3s);

    IF tOpen.Q THEN
        OpenOut := FALSE;
        Busy := FALSE;
        Done := TRUE;
        OpenedSim := TRUE;
        ClosedSim := FALSE;
        tOpen(IN := FALSE);
        State := 0;
    END_IF

END_CASE

END_FUNCTION_BLOCK

// ---- POUs/FB_RollerDoor.TcPOU
FUNCTION_BLOCK FB_RollerDoor
VAR_INPUT
    CloseCmd   : BOOL;
    OpenCmd    : BOOL;
END_VAR

VAR_OUTPUT
    CloseOut   : BOOL;
    OpenOut    : BOOL;
    Done       : BOOL;
    Busy       : BOOL;
    ClosedSim  : BOOL;
    OpenedSim  : BOOL;
END_VAR

VAR
    State   : INT := 0;
    tClose  : TON;
    tOpen   : TON;
END_VAR

CASE State OF

0: // Idle
    Done := FALSE;
    Busy := FALSE;
    CloseOut := FALSE;
    OpenOut := FALSE;

    tClose(IN := FALSE);
    tOpen(IN := FALSE);

    IF CloseCmd THEN
        State := 10;
    ELSIF OpenCmd THEN
        State := 20;
    END_IF


10: // Closing
    Busy := TRUE;
    CloseOut := TRUE;

    tClose(IN := TRUE, PT := T#4S);

    IF tClose.Q THEN
        CloseOut := FALSE;
        Busy := FALSE;
        Done := TRUE;
        ClosedSim := TRUE;
        OpenedSim := FALSE;
        tClose(IN := FALSE);
        State := 0;
    END_IF


20: // Opening
    Busy := TRUE;
    OpenOut := TRUE;

    tOpen(IN := TRUE, PT := T#4S);

    IF tOpen.Q THEN
        OpenOut := FALSE;
        Busy := FALSE;
        Done := TRUE;
        OpenedSim := TRUE;
        ClosedSim := FALSE;
        tOpen(IN := FALSE);
        State := 0;
    END_IF

END_CASE

END_FUNCTION_BLOCK

// ---- POUs/FB_Trunnion.TcPOU
FUNCTION_BLOCK FB_Trunnion
VAR_INPUT
    To0  : BOOL;
    To50 : BOOL;
END_VAR

VAR_OUTPUT
    CmdTo0  : BOOL;
    CmdTo50 : BOOL;
    Busy    : BOOL;
    At0     : BOOL;
    At50    : BOOL;
END_VAR

VAR
    State : INT := 0;
    tMove : TON;
END_VAR

CASE State OF

0:
    Busy := FALSE;
    CmdTo0 := FALSE;
    CmdTo50 := FALSE;
    At0 := TRUE;
    At50 := FALSE;
    tMove(IN := FALSE);

    IF To50 THEN State := 10;
    END_IF

10:
    Busy := TRUE;
    CmdTo50 := TRUE;
    At0 := FALSE;

    tMove(IN := TRUE, PT := T#5s);

    IF tMove.Q THEN
        CmdTo50 := FALSE;
        Busy := FALSE;
        At50 := TRUE;
        tMove(IN := FALSE);
        State := 20;
    END_IF

20:
    At50 := TRUE;

    IF To0 THEN State := 30;
    END_IF

30:
    Busy := TRUE;
    CmdTo0 := TRUE;
    At50 := FALSE;

    tMove(IN := TRUE, PT := T#5s);

    IF tMove.Q THEN
        CmdTo0 := FALSE;
        Busy := FALSE;
        At0 := TRUE;
        tMove(IN := FALSE);
        State := 0;
    END_IF

END_CASE

END_FUNCTION_BLOCK

// ---- POUs/FB_TurnTable.TcPOU
FUNCTION_BLOCK FB_Turntable
VAR_INPUT
    To180 : BOOL;
    To0   : BOOL;
END_VAR

VAR_OUTPUT
    Cmd180 : BOOL;
    Cmd0   : BOOL;
    Busy   : BOOL;
    At0    : BOOL;
    At180  : BOOL;
END_VAR

VAR
    State : INT := 0;
    tMove : TON;
END_VAR


CASE State OF

0:
    Busy := FALSE;
    Cmd180 := FALSE;
    Cmd0 := FALSE;

    At0 := TRUE;
    At180 := FALSE;

    tMove(IN := FALSE);

    IF To180 THEN State := 10;
    END_IF

10:
    Busy := TRUE;
    Cmd180 := TRUE;
    At0 := FALSE;

    tMove(IN := TRUE, PT := T#10s);

    IF tMove.Q THEN
        Cmd180 := FALSE;
        Busy := FALSE;
        At180 := TRUE;
        tMove(IN := FALSE);
        State := 20;
    END_IF

20:
    At180 := TRUE;

    IF To0 THEN State := 30;
    END_IF

30:
    Busy := TRUE;
    Cmd0 := TRUE;
    At180 := FALSE;

    tMove(IN := TRUE, PT := T#10s);

    IF tMove.Q THEN
        Cmd0 := FALSE;
        Busy := FALSE;
        At0 := TRUE;
        tMove(IN := FALSE);
        State := 0;
    END_IF

END_CASE

END_FUNCTION_BLOCK

// ---- POUs/FB_Robot.TcPOU
FUNCTION_BLOCK FB_Robot
VAR_INPUT
    StartWeld1 : BOOL;
    StartWeld2 : BOOL;
END_VAR

VAR_OUTPUT
    Weld1Active : BOOL;
    Weld2Active : BOOL;
    Busy        : BOOL;
    WeldDone1   : BOOL;
    WeldDone2   : BOOL;
END_VAR

VAR
    State   : INT := 0;
    tWeld   : TON;

    rTrig1  : R_TRIG;   // Rising edge for Weld1
    rTrig2  : R_TRIG;   // Rising edge for Weld2
END_VAR


// Edge detection (prevents continuous retrigger)
rTrig1(CLK := StartWeld1);
rTrig2(CLK := StartWeld2);


CASE State OF

//--------------------------------------------------
// 0: IDLE
//--------------------------------------------------
0:
    Busy := FALSE;

    Weld1Active := FALSE;
    Weld2Active := FALSE;

    WeldDone1 := FALSE;
    WeldDone2 := FALSE;

    tWeld(IN := FALSE);

    // Start only on rising edge
    IF rTrig1.Q THEN
        State := 10;
    ELSIF rTrig2.Q THEN
        State := 20;
    END_IF


//--------------------------------------------------
// 10: WELD 1
//--------------------------------------------------
10:
    Busy := TRUE;
    Weld1Active := TRUE;

    tWeld(IN := TRUE, PT := T#6s);

    IF tWeld.Q THEN
        Weld1Active := FALSE;
        WeldDone1 := TRUE;

        Busy := FALSE;
        tWeld(IN := FALSE);

        State := 0;
    END_IF


//--------------------------------------------------
// 20: WELD 2
//--------------------------------------------------
20:
    Busy := TRUE;
    Weld2Active := TRUE;

    tWeld(IN := TRUE, PT := T#6s);

    IF tWeld.Q THEN
        Weld2Active := FALSE;
        WeldDone2 := TRUE;

        Busy := FALSE;
        tWeld(IN := FALSE);

        State := 0;
    END_IF

END_CASE

END_FUNCTION_BLOCK

// ---- POUs/FB_Robot_MH.TcPOU
FUNCTION_BLOCK FB_Robot_MH
VAR_INPUT
    ClearToPick1 : BOOL;
    ClearToPick2 : BOOL;
END_VAR

VAR_OUTPUT
    Pick1Active : BOOL;
    Pick2Active : BOOL;
    Busy        : BOOL;
    Pick1Done1   : BOOL;
    Pick2Done2   : BOOL;
END_VAR

VAR
    State   : INT := 0;
    tPick   : TON;

    rTrig1  : R_TRIG;   // Rising edge for Weld1
    rTrig2  : R_TRIG;   // Rising edge for Weld2
END_VAR


// Edge detection (prevents continuous retrigger)
rTrig1(CLK := ClearToPick1);
rTrig2(CLK := ClearToPick2);


CASE State OF

//--------------------------------------------------
// 0: IDLE
//--------------------------------------------------
0:
    Busy := FALSE;

    Pick1Active := FALSE;
    Pick1Active := FALSE;

    Pick1Done1 := FALSE;
    Pick2Done2 := FALSE;

    tPick(IN := FALSE);

    // Start only on rising edge
    IF rTrig1.Q THEN
        State := 10;
    ELSIF rTrig2.Q THEN
        State := 20;
    END_IF


//--------------------------------------------------
// 10: WELD 1
//--------------------------------------------------
10:
    Busy := TRUE;
    Pick1Active := TRUE;

    tPick(IN := TRUE, PT := T#6S);

    IF tPick.Q THEN
        Pick1Active := FALSE;
        Pick1Done1 := TRUE;

        Busy := FALSE;
        tPick(IN := FALSE);

        State := 0;
    END_IF


//--------------------------------------------------
// 20: WELD 2
//--------------------------------------------------
20:
    Busy := TRUE;
    Pick2Active := TRUE;

    tPick(IN := TRUE, PT := T#6S);

    IF tPick.Q THEN
        Pick2Active := FALSE;
        Pick2Done2 := TRUE;

        Busy := FALSE;
        tPick(IN := FALSE);

        State := 0;
    END_IF

END_CASE

END_FUNCTION_BLOCK

// ---- GlobalTextList.TcGTLO
TEXTLIST GlobalTextList
  891 = '1'
  867 = '2'
  393 = '3'
  759 = '4'
  178 = 'AUTO'
  130 = 'Auto On'
  897 = 'CC1 Close'
  905 = 'CC1 Open'
  879 = 'CC2 Close'
  205 = 'CC2 Open'
  610 = 'CC3 Close'
  233 = 'CC3 Open'
  693 = 'CC4 Close'
  106 = 'CC4 Open'
  453 = 'CC5 Close'
  236 = 'CC5 Open'
  852 = 'CC6 Close'
  113 = 'CC6 Open'
  354 = 'Clamp1'
  11 = 'Clamp1 Close'
  699 = 'Clamp1 Open'
  151 = 'Clamp2 Close'
  123 = 'Clamp2 Open'
  930 = 'Clamp3 Close'
  841 = 'Clamp3 Open'
  900 = 'Clamp4 Close'
  265 = 'Clamp4 Open'
  253 = 'Cycle Start'
  972 = 'Cycle Start PB'
  607 = 'Done'
  653 = 'Door Close'
  298 = 'Door Closed'
  751 = 'Door Open'
  470 = 'Door Opened'
  725 = 'E-Stop'
  266 = 'FIX1- Manual'
  487 = 'FIX2- Manual'
  258 = 'LC'
  435 = 'MAN'
  349 = 'Manual On'
  510 = 'Manual Operations'
  425 = 'OP Box'
  828 = 'Oper. Box'
  121 = 'Operator Side-0'
  460 = 'Operator Side-180'
  766 = 'Part Pres1 '
  985 = 'Part Pres2'
  307 = 'Part Pres3'
  259 = 'Part Pres4 '
  346 = 'Robot  Pick 2 On'
  538 = 'Robot  Weld 2 On'
  737 = 'Robot 1 Weld On'
  356 = 'Robot 2 Weld On'
  513 = 'Robot Pick 1 Done'
  65 = 'Robot Pick 1 On'
  752 = 'Robot Pick 2 Done'
  419 = 'Robot Weld 1 Complete'
  924 = 'Robot Weld 1 Complte'
  931 = 'Robot Weld 1 Done'
  290 = 'Robot Weld 1 Done On'
  191 = 'Robot Weld 1 On'
  282 = 'Robot Weld 2 Done'
  769 = 'Robot Weld On'
  781 = 'Roll Door Close'
  842 = 'Trunn to 0'
  211 = 'Trunn to 180'
  77 = 'Trunn to 50'
  295 = 'Trunn1 to 0'
  52 = 'Trunn1 to 50'
  164 = 'Trunn2 to 0'
  102 = 'Trunn2 to 50'
  499 = 'Trunnion 0 Degree'
  278 = 'Trunnion 50 Degree'
  563 = 'Trunnion1 0 Degree'
  423 = 'Trunnion1 50 Degree'
  197 = 'Trunnion2 0 Degree'
  469 = 'Trunnion2 50 Degree'
  3 = 'TT to 0'
  20 = 'TT to 180'
  688 = 'Turntable 0 Degree'
  344 = 'Turntable 180 Degree'
  452 = 'Weld Comp 1'
  471 = 'Weld Comp 2'
  990 = 'Weld Side-180'
END_TEXTLIST

// ---- POUs/TextList_State1.TcTLO
TEXTLIST TextList_State1
  0 = 'Wait for Door Open..'
  10 = 'Wait For Part 1 Load and Cycle Start...'
  20 = 'Door Closing...'
  30 = 'Clamp CC1 CC3 CC5 Closing...'
  40 = 'Trunmion is Moving 0 to 50 Degree for Load 2'
  50 = 'Door Opening...'
  60 = 'Wait For Part 2 Load and Cycle Start...'
  70 = 'Clamp CC2 CC4 CC6 Closing..'
  80 = 'Door Closing...'
  90 = 'Trunmion is Moving 50 to 0 Degree...'
  100 = 'Turn Table Moving 0 to 180 Degree for weld Position...'
  110 = 'Robot Start....Waiting for Weld Complete 1....'
  120 = 'Trunmion is Moving 0 to 50 Degree for Weld 2...'
  130 = 'Robot Start....Waiting for Weld Complete 2....'
  140 = 'Clamp CC1 CC3 CC5 Opening...'
  150 = 'Robot Clear To Pick....Waiting for Pick Complete 1....'
  160 = 'Trunmion is Moving 0 Degree for Pick 2...'
  170 = 'Clamp CC2 CC4 CC6 Opening...'
  180 = 'Robot Clear To Pick....Waiting for Pick Complete 2....'
   = ''
END_TEXTLIST

// ---- POUs/TextList_State2.TcTLO
TEXTLIST TextList_State2
  0 = 'Wait for Door Open..'
  10 = 'Wait For Part 1 Load and Cycle Start...'
  20 = 'Door Closing...'
  30 = 'Clamp CC1 CC3 CC5 Closing...'
  40 = 'Trunmion is Moving 0 to 50 Degree for Load 2'
  50 = 'Door Opening...'
  60 = 'Wait For Part 2 Load and Cycle Start...'
  70 = 'Clamp CC2 CC4 CC6 Closing..'
  80 = 'Door Closing...'
  90 = 'Trunmion is Moving 50 to 0 Degree...'
  100 = 'Turn Table Moving 0 to 180 Degree for weld Position...'
  110 = 'Robot Start....Waiting for Weld Complete 1....'
  120 = 'Trunmion is Moving 0 to 50 Degree for Weld 2...'
  130 = 'Robot Start....Waiting for Weld Complete 2....'
  140 = 'Clamp CC1 CC3 CC5 Opening...'
  150 = 'Robot Clear To Pick....Waiting for Pick Complete 1....'
  160 = 'Trunmion is Moving 0 Degree for Pick 2...'
  170 = 'Clamp CC2 CC4 CC6 Opening...'
  180 = 'Robot Clear To Pick....Waiting for Pick Complete 2....'
   = ''
END_TEXTLIST

// ---- POUs/Visualization.TcVIS
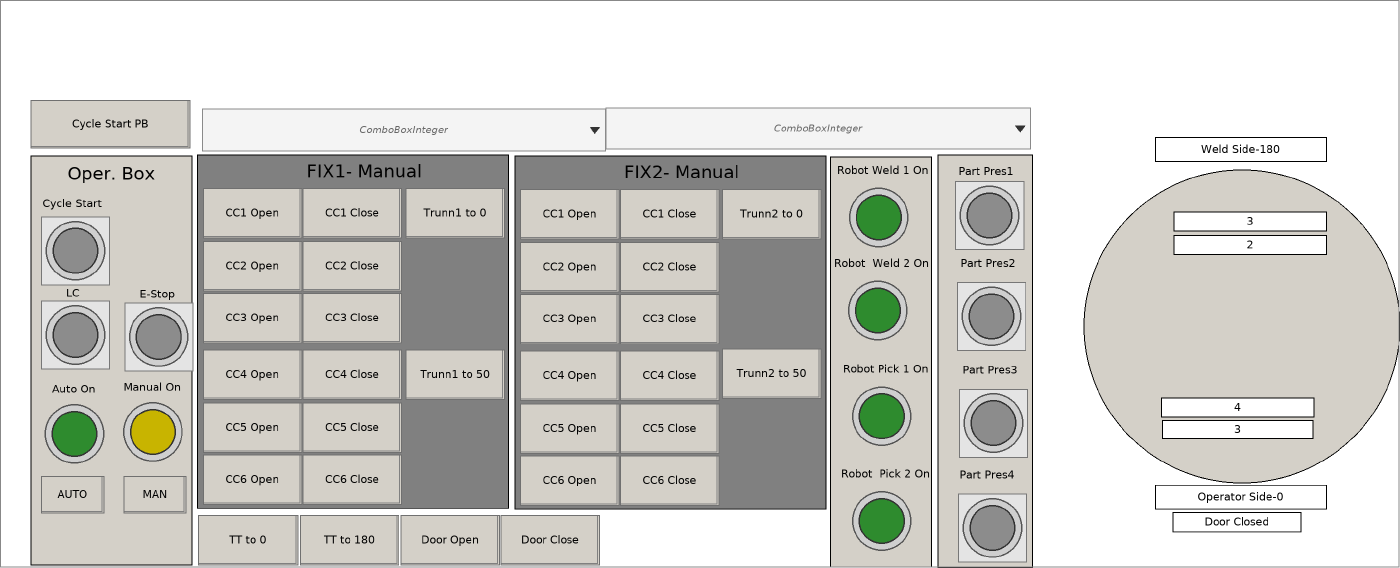
VISUALIZATION Visualization  // 1429x580
    Rectangle (957,158 97x422)
    Rectangle (847,160 104x419)
    Rectangle (31,159 165x418)
    PushSwitchLed (973,185 74x70), variable: MAIN.PartPresent1, behaviour: TOGGLE, style: Switch-PushSwitchLed-Gray
    Label (964,160 89x30), "Part Pres1"
    PushSwitchLed (40,221 74x70), variable: MAIN.CycleStart, behaviour: TOGGLE, style: Switch-PushSwitchLed-Gray
    Label (29,193 90x30), "Cycle Start"
    PushSwitchLed (975,288 74x70), variable: MAIN.PartPresent2, behaviour: TOGGLE, style: Switch-PushSwitchLed-Gray
    Label (964,254 89x30), "Part Pres2"
    Button (42,486 64x38), "AUTO", text variable: MAIN.HMI_Auto, colour toggle: MAIN.HMI_Auto
        tap MAIN.HMI_Auto
    PushSwitchLed (977,397 74x70), variable: MAIN.PartPresent3, behaviour: TOGGLE, style: Switch-PushSwitchLed-Gray
    PushSwitchLed (976,504 74x70), variable: MAIN.PartPresent4, behaviour: TOGGLE, style: Switch-PushSwitchLed-Gray
    Label (965,470 89x30), "Part Pres4"
    Label (966,363 89x30), "Part Pres3"
    PushSwitchLed (125,309 74x70), variable: MAIN.EmergencyStop, behaviour: TOGGLE, style: Switch-PushSwitchLed-Gray
    Label (116,288 89x25), "E-Stop"
    Label (30,287 89x25), "LC"
    PushSwitchLed (40,307 74x70), variable: MAIN.LightCurtainOK, behaviour: TOGGLE, style: Switch-PushSwitchLed-Gray
    Lamp1 (862,187 70x70), variable: MAIN.Robot1.Weld1Active, style: Lamp-Lamp1-Green
    Label (850,159 102x30), "Robot Weld 1 On"
    Lamp1 (861,282 70x70), variable: MAIN.Robot1.Weld2Active, style: Lamp-Lamp1-Green
    Label (849,254 102x30), "Robot Weld 2 On"
    Lamp1 (41,408 70x70), variable: MAIN.ModeMgr.AutoMode, style: Lamp-Lamp1-Green
    Label (31,385 89x25), "Auto On"
    Button (126,486 64x38), "MAN", text variable: MAIN.HMI_Manual, colour toggle: MAIN.HMI_Manual
        tap MAIN.HMI_Manual
    ComboBoxInteger (206,111 412x43), variable: MAIN.AutoSeq.State1, text list: 'TextList_State1'
    ComboBoxInteger (618,110 434x42), variable: MAIN.AutoSeq.State2, text list: 'TextList_State2'
    Lamp1 (121,406 70x70), variable: MAIN.ModeMgr.ManualMode, style: Lamp-Lamp1-Yellow
    Label (111,383 89x25), "Manual On"
    Label (8,166 211x23), "Oper. Box"
    Ellipse (1106,173 323x320)
    Rectangle (1186,429 154x19), "1", colour toggle: MAIN.Trunnion1.At0, invisible if: MAIN.Turntable.At180
    Rectangle (1185,406 156x20), "2", colour toggle: MAIN.Trunnion1.At50, invisible if: MAIN.Turntable.At180
    Rectangle (1186,429 154x19), "3", colour toggle: MAIN.Trunnion2.At0, invisible if: MAIN.Turntable.At0
    Rectangle (1185,406 156x20), "4", colour toggle: MAIN.Trunnion2.At50, invisible if: MAIN.Turntable.At0
    Rectangle (1198,240 156x20), "4", colour toggle: MAIN.Trunnion2.At50, invisible if: MAIN.Turntable.At180
    Rectangle (1198,216 156x20), "1", colour toggle: MAIN.Trunnion1.At0, invisible if: MAIN.Turntable.At0
    Rectangle (1198,240 156x20), "2", colour toggle: MAIN.Trunnion1.At50, invisible if: MAIN.Turntable.At0
    Rectangle (1198,216 156x20), "3", colour toggle: MAIN.Trunnion2.At0, invisible if: MAIN.Turntable.At180
    Rectangle (1179,140 175x25), "Weld Side-180", colour toggle: MAIN.Turntable.At180
    Rectangle (1179,495 175x25), "Operator Side-0", colour toggle: MAIN.Turntable.At0
    Rectangle (1197,523 131x20), "Door Opened", colour toggle: MAIN.RollerDoor1.OpenedSim, invisible if: MAIN.RollerDoor1.ClosedSim
    Rectangle (1197,523 131x20), "Door Closed", colour toggle: MAIN.RollerDoor1.ClosedSim, invisible if: MAIN.RollerDoor1.OpenedSim
    Button (31,102 163x49), "Cycle Start PB", text variable: MAIN.CycleStart, colour toggle: MAIN.CycleStart
        tap MAIN.CycleStart
    Rectangle (201,158 318x361)
    Button (202,526 102x51), "TT to 0", text variable: MAIN.Turntable.At0, colour toggle: MAIN.Turntable.At0
        tap MAIN.ManTT0
    Button (306,526 101x51), "TT to 180", text variable: MAIN.Turntable.At180, colour toggle: MAIN.Turntable.At180
        tap MAIN.ManTT180
    Button (414,192 101x51), "Trunn1 to 0", text variable: MAIN.Trunnion1.At0, colour toggle: MAIN.Trunnion1.At0
        tap MAIN.ManTrn10
    Button (414,357 101x51), "Trunn1 to 50", text variable: MAIN.Trunnion1.At50, colour toggle: MAIN.Trunnion1.At50
        tap MAIN.ManTrn150
    Button (309,192 101x51), "CC1 Close", text variable: MAIN.Fixture_1_CC1.ClosedSim, colour toggle: MAIN.Fixture_1_CC1.ClosedSim
        tap MAIN.Fixture_1_ManCC1Close
    Button (207,192 101x51), "CC1 Open", text variable: MAIN.Fixture_1_CC1.OpenedSim, colour toggle: MAIN.Fixture_1_CC1.OpenedSim
        tap MAIN.Fixture_1_ManCC1Open
    Label (242,155 260x40), "FIX1- Manual"
    Button (409,526 101x51), "Door Open", text variable: MAIN.RollerDoor1.OpenedSim, colour toggle: MAIN.RollerDoor1.OpenedSim
        tap MAIN.ManRollerDoor1Open
    Button (511,526 101x51), "Door Close", text variable: MAIN.RollerDoor1.ClosedSim, colour toggle: MAIN.RollerDoor1.ClosedSim
        tap MAIN.ManRollerDoor1Close
    Lamp1 (865,390 70x70), variable: MAIN.Robot2.Pick1Active, style: Lamp-Lamp1-Green
    Label (853,362 102x30), "Robot Pick 1 On"
    Lamp1 (865,497 70x70), variable: MAIN.Robot2.Pick2Active, style: Lamp-Lamp1-Green
    Label (853,469 102x30), "Robot Pick 2 On"
    Button (309,246 101x51), "CC2 Close", text variable: MAIN.Fixture_1_CC2.ClosedSim, colour toggle: MAIN.Fixture_1_CC2.ClosedSim
        tap MAIN.Fixture_1_ManCC2Close
    Button (207,246 101x51), "CC2 Open", text variable: MAIN.Fixture_1_CC2.OpenedSim, colour toggle: MAIN.Fixture_1_CC2.OpenedSim
        tap MAIN.Fixture_1_ManCC2Open
    Button (207,299 101x51), "CC3 Open", text variable: MAIN.Fixture_1_CC3.OpenedSim, colour toggle: MAIN.Fixture_1_CC3.OpenedSim
        tap MAIN.Fixture_1_ManCC3Open
    Button (309,299 101x51), "CC3 Close", text variable: MAIN.Fixture_1_CC3.ClosedSim, colour toggle: MAIN.Fixture_1_CC3.ClosedSim
        tap MAIN.Fixture_1_ManCC3Close
    Button (207,357 101x51), "CC4 Open", text variable: MAIN.Fixture_1_CC4.OpenedSim, colour toggle: MAIN.Fixture_1_CC4.OpenedSim
        tap MAIN.Fixture_1_ManCC4Open
    Button (309,357 101x51), "CC4 Close", text variable: MAIN.Fixture_1_CC4.ClosedSim, colour toggle: MAIN.Fixture_1_CC4.ClosedSim
        tap MAIN.Fixture_1_ManCC4Close
    Button (309,411 101x51), "CC5 Close", text variable: MAIN.Fixture_1_CC5.ClosedSim, colour toggle: MAIN.Fixture_1_CC5.ClosedSim
        tap MAIN.Fixture_1_ManCC5Close
    Button (207,411 101x51), "CC5 Open", text variable: MAIN.Fixture_1_CC5.OpenedSim, colour toggle: MAIN.Fixture_1_CC5.OpenedSim
        tap MAIN.Fixture_1_ManCC5Open
    Button (207,464 101x51), "CC6 Open", text variable: MAIN.Fixture_1_CC6.OpenedSim, colour toggle: MAIN.Fixture_1_CC6.OpenedSim
        tap MAIN.Fixture_1_ManCC6Open
    Button (309,464 101x51), "CC6 Close", text variable: MAIN.Fixture_1_CC6.ClosedSim, colour toggle: MAIN.Fixture_1_CC6.ClosedSim
        tap MAIN.Fixture_1_ManCC6Close
    Rectangle (525,159 318x361)
    Button (633,193 101x51), "CC1 Close", text variable: MAIN.Fixture_2_CC1.ClosedSim, colour toggle: MAIN.Fixture_2_CC1.ClosedSim
        tap MAIN.Fixture_2_ManCC1Close
    Button (531,193 101x51), "CC1 Open", text variable: MAIN.Fixture_2_CC1.OpenedSim, colour toggle: MAIN.Fixture_2_CC1.OpenedSim
        tap MAIN.Fixture_2_ManCC1Open
    Label (566,156 260x40), "FIX2- Manual"
    Button (633,247 101x51), "CC2 Close", text variable: MAIN.Fixture_2_CC2.ClosedSim, colour toggle: MAIN.Fixture_2_CC2.ClosedSim
        tap MAIN.Fixture_2_ManCC2Close
    Button (531,247 101x51), "CC2 Open", text variable: MAIN.Fixture_2_CC2.OpenedSim, colour toggle: MAIN.Fixture_2_CC2.OpenedSim
        tap MAIN.Fixture_2_ManCC2Open
    Button (531,300 101x51), "CC3 Open", text variable: MAIN.Fixture_2_CC3.OpenedSim, colour toggle: MAIN.Fixture_2_CC3.OpenedSim
        tap MAIN.Fixture_2_ManCC3Open
    Button (633,300 101x51), "CC3 Close", text variable: MAIN.Fixture_2_CC3.ClosedSim, colour toggle: MAIN.Fixture_2_CC3.ClosedSim
        tap MAIN.Fixture_2_ManCC3Close
    Button (531,358 101x51), "CC4 Open", text variable: MAIN.Fixture_2_CC4.OpenedSim, colour toggle: MAIN.Fixture_2_CC4.OpenedSim
        tap MAIN.Fixture_2_ManCC4Open
    Button (633,358 101x51), "CC4 Close", text variable: MAIN.Fixture_2_CC4.ClosedSim, colour toggle: MAIN.Fixture_2_CC4.ClosedSim
        tap MAIN.Fixture_2_ManCC4Close
    Button (633,412 101x51), "CC5 Close", text variable: MAIN.Fixture_2_CC5.ClosedSim, colour toggle: MAIN.Fixture_2_CC5.ClosedSim
        tap MAIN.Fixture_2_ManCC5Close
    Button (531,412 101x51), "CC5 Open", text variable: MAIN.Fixture_2_CC5.OpenedSim, colour toggle: MAIN.Fixture_2_CC5.OpenedSim
        tap MAIN.Fixture_2_ManCC5Open
    Button (531,465 101x51), "CC6 Open", text variable: MAIN.Fixture_2_CC6.OpenedSim, colour toggle: MAIN.Fixture_2_CC6.OpenedSim
        tap MAIN.Fixture_2_ManCC6Open
    Button (633,465 101x51), "CC6 Close", text variable: MAIN.Fixture_2_CC6.ClosedSim, colour toggle: MAIN.Fixture_2_CC6.ClosedSim
        tap MAIN.Fixture_2_ManCC6Close
    Button (737,193 101x51), "Trunn2 to 0", text variable: MAIN.Trunnion2.At0, colour toggle: MAIN.Trunnion2.At0
        tap MAIN.ManTrn20
    Button (737,356 101x51), "Trunn2 to 50", text variable: MAIN.Trunnion2.At50, colour toggle: MAIN.Trunnion2.At50
        tap MAIN.ManTrn250
END_VISUALIZATION
